// TIA Portal V20 export
TYPE "HMI_OpDi03"
   STRUCT
      SetOp1 : Bool;   // Operator Digital Input 1
      SetOp2 : Bool;   // Operator Digital Input 2
      SetOp3 : Bool;   // Operator Digital Input 3
      SetLi1 : Bool;   // Linkable Digital Input 1
      SetLi2 : Bool;   // Linkable Digital Input 2
      SetLi3 : Bool;   // Linkable Digital Input 3
      RstOut : Bool;   // Reset Output
      Intlock : Bool := true;   // 0=Interlocked, 1=Not Interlocked
      Intlock_ST : Byte := BYTE#16#FF;   // Intlock Signal Status
      OnOp : Bool;   // 1=On Mode: On Mode by Operator
      OosOp : Bool;   // 1=Oos Mode: Oos Mode by Operator
      OS_PermOut { ExternalWritable := 'False'} : DWord;   // Operator Permission: Output for OS
      OS_PermLog { ExternalWritable := 'False'} : DWord;   // Operator Permission: Output for OS
      OpSt_Out { ExternalWritable := 'False'} : DWord;   // Enabled operator stations
      ST_Worst { ExternalWritable := 'False'} : Byte;   // Worst Signal Status
      Status { ExternalWritable := 'False'} : DWord;   // Status Word
   END_STRUCT;
END_TYPE
